// LS Electric XG5000 project: Sorting_Station
// PLC LSPLC

PROGRAM NewProgram (task: 스캔 프로그램)

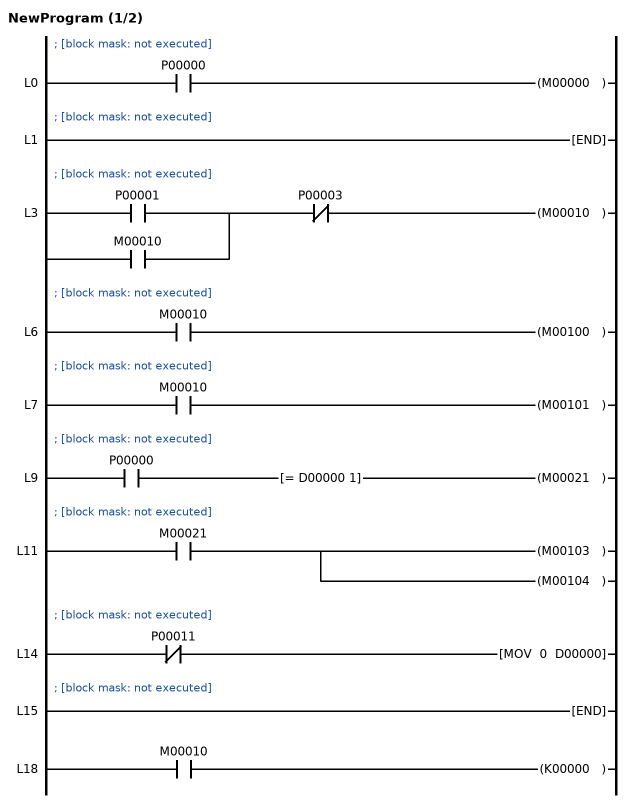
; L0 (block mask: not executed)
LOAD      P00000
OUT       M00000
; L1 (block mask: not executed)
END
; L3 (block mask: not executed)
LOAD      P00001
OR        M00010
AND NOT   P00003
OUT       M00010
; L6 (block mask: not executed)
LOAD      M00010
OUT       M00100
; L7 (block mask: not executed)
LOAD      M00010
OUT       M00101
; L9 (block mask: not executed)
LOAD      P00000
AND=      D00000 1
OUT       M00021
; L11 (block mask: not executed)
LOAD      M00021
OUT       M00103
OUT       M00104
; L14 (block mask: not executed)
LOAD NOT  P00011
MOV       0 D00000
; L15 (block mask: not executed)
END
; L18
LOAD      M00010
OUT       K00000

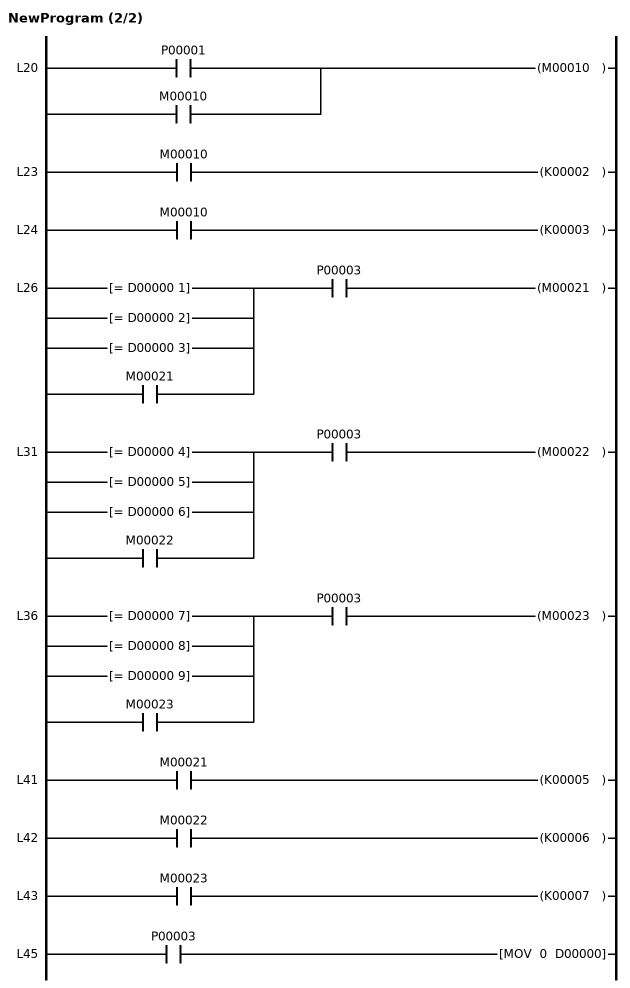
; L20
LOAD      P00001
OR        M00010
OUT       M00010
; L23
LOAD      M00010
OUT       K00002
; L24
LOAD      M00010
OUT       K00003
; L26
LOAD=     D00000 1
OR=       D00000 2
OR=       D00000 3
OR        M00021
AND       P00003
OUT       M00021
; L31
LOAD=     D00000 4
OR=       D00000 5
OR=       D00000 6
OR        M00022
AND       P00003
OUT       M00022
; L36
LOAD=     D00000 7
OR=       D00000 8
OR=       D00000 9
OR        M00023
AND       P00003
OUT       M00023
; L41
LOAD      M00021
OUT       K00005
; L42
LOAD      M00022
OUT       K00006
; L43
LOAD      M00023
OUT       K00007
; L45
LOAD      P00003
MOV       0 D00000